FUNCTION_BLOCK F_TO_C_CONV (* Basic FB with empty ECC *)
  (* Standard: 61499-2 *)
  (* Version 1.0, 2020-10-20, chong *)
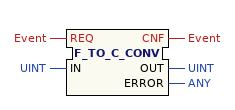
  EVENT_INPUT
    REQ;
  END_EVENT
  EVENT_OUTPUT
    CNF;
  END_EVENT
  VAR_INPUT
    IN : UINT;
  END_VAR
  VAR_OUTPUT
    OUT : UINT;
    ERROR : ANY;
  END_VAR
  EC_STATES
    START; (* Initial State *)
  END_STATES
END_FUNCTION_BLOCK
